TYPE ST_eChillerDefaultParameters :
STRUCT
	aSetPointLimitsTemperature : ARRAY[1..2] OF REAL;
END_STRUCT
END_TYPE

(* stored: Version 1.1.0.1, ProductVersion 3.1.4024.9
   DUT ST_eChillerDefaultParameters: Id {5e1708f4-4b24-4710-a81f-ab3e89a27f17} *)
